// TIA Portal V20 export
FUNCTION_BLOCK "FB_OPC_State"   // FB75, SCL
{ S7_Optimized_Access := 'TRUE' }
// stored: MemoryReserve 100, SetENOAutomatically false
   VAR
      sAutoReq : Bool;
      sSemiAutoReq : Bool;
      sManuReq : Bool;
      sRT_AutoReq : R_TRIG;
      sRT_SemiAutoReq : R_TRIG;
      sRT_ManuReq : R_TRIG;
   END_VAR
   VAR CONSTANT
      AUTO : Byte := 1;
      SEMI_AUTO : Byte := 2;
      MANU : Byte := 3;
      UNDEFINED : Byte := 0;
   END_VAR
BEGIN
   REGION Description header 
       //==================================================================================
       // POSALUX Swiss SA / (C) Copyright 2024
       //----------------------------------------------------------------------------------
       // Title: 
       // Comment/Function: 
       //
       // Author: Fabien WALDT
       // Engineering: TIA Portal v20
       //----------------------------------------------------------------------------------
       // Change log table:
       // Version  | Date     | Expert in charge | Changes applied
       // ---------|----------|------------------|------------------------------------
       // 00.00.01 | 20260130 | WFA              | First released version
       // ==================================================================================
   END_REGION

   REGION Current
       // CanLockDoor
       "DB_OPC_Machine".State.Current.CanLockDoor := "LBP_ModeGroup".E_JOG
       AND "DB_DigitalInputs".sFrontDoorClosed.sSWStatus;

       // CanUnlockDoor
       "DB_OPC_Machine".State.Current.CanUnlockDoor := "LBP_ModeGroup".E_JOG
       AND "DB_DigitalInputs".sFrontDoorLocked.sSWStatus;

       // LoadingMode
       // 1 = Auto
       // 2 = Semi Auto
       // 3 = Manu 
       IF "DB_WorkingModes".sAuto THEN
           "DB_OPC_Machine".State.Current.LoadingMode := #AUTO;
       ELSIF "DB_WorkingModes".sSemiAuto THEN
           "DB_OPC_Machine".State.Current.LoadingMode := #SEMI_AUTO;
       ELSIF "DB_WorkingModes".sManu THEN
           "DB_OPC_Machine".State.Current.LoadingMode := #MANU;
       ELSE
           "DB_OPC_Machine".State.Current.LoadingMode := #UNDEFINED;
       END_IF;

       // IsDoorLocked
       "DB_OPC_Machine".State.Current.IsDoorLocked := "DB_DigitalInputs".sFrontDoorLocked.sSWStatus;

       // IsEmptying
       "DB_OPC_Machine".State.Current.IsEmptying := "DB_WorkingModes".sEmptying;

       // IsInitialized
       "DB_OPC_Machine".State.Current.IsInitialized := "DB_PowerOn".sMachineReadySoft;

       // IsRunning
       "DB_OPC_Machine".State.Current.IsRunning := "LBP_Chan1".E_ProgRunning;
   END_REGION

   REGION
       // Request Change Mode
       IF "DB_OPC_Machine".State.Requests.LoadingMode.RequestChangeMode THEN
           IF "DB_OPC_Machine".State.Requests.LoadingMode.TargetMode = #AUTO THEN
               #sAutoReq := TRUE;
           ELSIF "DB_OPC_Machine".State.Requests.LoadingMode.TargetMode = #SEMI_AUTO THEN
               #sSemiAutoReq := TRUE;
           ELSIF "DB_OPC_Machine".State.Requests.LoadingMode.TargetMode = #MANU THEN
               #sManuReq := TRUE;
           END_IF;
           "DB_OPC_Machine".State.Requests.LoadingMode.RequestChangeMode := FALSE;
           "DB_OPC_Machine".State.Requests.LoadingMode.TargetMode := #UNDEFINED;
       END_IF;

       #sRT_AutoReq(CLK := #sAutoReq);
       #sRT_SemiAutoReq(CLK := #sSemiAutoReq);
       #sRT_ManuReq(CLK := #sManuReq);

       // Request Lock Door
       IF "DB_OPC_Machine".State.Requests.RequestLockDoor THEN
           "DB_HMISetting".LockDoorReq := TRUE;
           "DB_OPC_Machine".State.Requests.RequestLockDoor := FALSE;
       END_IF;

       // Request Start Auto
       IF "DB_OPC_Machine".State.Requests.RequestStartAuto THEN
           "DB_HMISetting".StartAutoReq := TRUE;
           "DB_OPC_Machine".State.Requests.RequestStartAuto := FALSE;
       END_IF;

       // Request Start Emptying
       IF "DB_OPC_Machine".State.Requests.RequestStartEmptying THEN
           "DB_HMISetting".WorkingMode.EmptyingReq := TRUE;
           "DB_OPC_Machine".State.Requests.RequestStartEmptying := FALSE;
       END_IF;

       // Request Stop Auto
       IF "DB_OPC_Machine".State.Requests.RequestStopAuto THEN
           "DB_HMISetting".StopAutoReq := TRUE;
           "DB_OPC_Machine".State.Requests.RequestStopAuto := FALSE;
       END_IF;

       // Request Stop Emptying (Back to Normal Mode)
       IF "DB_OPC_Machine".State.Requests.RequestStopEmptying THEN
           "DB_HMISetting".WorkingMode.EmptyingReq := FALSE;
       END_IF;
       "DB_OPC_Machine".State.Requests.RequestStopEmptying := FALSE;

       // Request Unlock Door
       IF "DB_OPC_Machine".State.Requests.RequestUnlockDoor THEN
           "DB_HMISetting".UnlockDoorReq := TRUE;
           "DB_OPC_Machine".State.Requests.RequestUnlockDoor := FALSE;
       END_IF;
   END_REGION

   REGION CNCMode
       IF "LBP_ModeGroup".E_AUTO THEN
           "DB_OPC_Machine".State.Current.CncMode := 1;
       ELSIF "LBP_ModeGroup".E_JOG THEN
           "DB_OPC_Machine".State.Current.CncMode := 2;
       ELSIF "LBP_ModeGroup".E_MDA THEN
           "DB_OPC_Machine".State.Current.CncMode := 3;
       ELSE
           "DB_OPC_Machine".State.Current.CncMode := 0;
       END_IF;
   END_REGION

   REGION MachineOverride
       "DB_OPC_Machine".State.Current.MachineOverride := "DB_FeedOverride".oFeedOverride;
   END_REGION
END_FUNCTION_BLOCK
